FUNCTION_BLOCK FB_CommandTest EXTENDS TcUnit.FB_TestSuite
VAR
	sText			: STRING;
	iCounter		: INT;
END_VAR


T01_TestPoleceniaProstego ();
T02_TestPoleceniaZlozonego ();

METHOD PUBLIC MetodaDlaPolecenbiaProstego : bool
VAR_INPUT
END_VAR
THIS^.sText := 'jestem w tej metodzie';
iCounter := iCounter + 1;
MetodaDlaPolecenbiaProstego	:= FALSE;
END_METHOD

METHOD PROTECTED T01_TestPoleceniaProstego
VAR_INPUT
END_VAR
IF (TcUnit.TEST_ORDERED ('T01_TestPoleceniaProstego')) THEN
	GVL.fbCommandEasy.Test ();
	AssertTrue (Condition := GVL.fbCommandEasy.IsStatus (), 	Message := 'T01a - Bledny status');
	AssertFalse (Condition := GVL.fbCommandEasy.IsBusy (),		Message := 'T01b - Bledny stan');
	GVL.fbCommandEasy.Execute ();
	GVL.fbCommandEasy.Test ();
	AssertFalse (Condition := GVL.fbCommandEasy.IsStatus (), 	Message := 'T02a - Bledny status');
	AssertTrue (Condition := GVL.fbCommandEasy.IsBusy (),		Message := 'T02b - Bledny stan');
	
	GVL.fbCommandEasy.OperationExecute ();
	GVL.fbCommandEasy.Operation (bIN := MetodaDlaPolecenbiaProstego ());
	
	AssertTrue (Condition := GVL.fbCommandEasy.IsFirstCycle (),Message := 'T03a - Bledny stan pierwszego przejscia');
	AssertTrue (Condition := GVL.fbCommandEasy.IsLastCycle (),	Message := 'T03b - Bledny stan ostatniego przejscia');
	
	GVL.fbCommandEasy.OperationExecute ();
	
	AssertFalse (Condition := GVL.fbCommandEasy.IsFirstCycle (),	Message := 'T04a - Bledny stan pierwszego przejscia');
	AssertFalse (Condition := GVL.fbCommandEasy.IsLastCycle (),		Message := 'T04b - Bledny stan ostatniego przejscia');

	GVL.fbCommandEasy.OperationExecute ();
	
	AssertFalse (Condition := GVL.fbCommandEasy.IsLastCycle (),	Message := 'T05a - Bledny stan pierwszego przejscia');
	AssertTrue (Condition := GVL.fbCommandEasy.IsStatus (),		Message := 'T05b - Bledny stan statusy');
	
	TcUnit.TEST_FINISHED ();
END_IF
END_METHOD

METHOD PROTECTED T02_TestPoleceniaZlozonego : BOOL

VAR
	bResult: BOOL;
END_VAR
IF (TcUnit.TEST_ORDERED ('T02_TestPolecenia')) THEN
	GVL.fbCommand.Test ();
	AssertTrue (Condition := GVL.fbCommand.IsStatus (), 	Message := 'T01a - Bledny status');
	AssertFalse (Condition := GVL.fbCommand.IsBusy (),		Message := 'T01b - Bledny stan');
	
	GVL.fbCommand.Execute ();
	GVL.fbCommand.Test ();
	AssertFalse (Condition := GVL.fbCommand.IsStatus (), 	Message := 'T02a - Bledny status');
	AssertTrue (Condition := GVL.fbCommand.IsBusy (),		Message := 'T02b - Bledny stan');
	
	IF (GVL.fbCommand.OperationExecute ()) THEN;
		bResult				:= TRUE;
		GVL.fbCommand.Operation (bIN := GVL.fbCommand.CyklTestu ());
	ELSE
		bResult				:= FALSE;
	END_IF
	AssertTrue (Condition := GVL.fbCommand.IsFirstCycle (),Message := 'T03a - Bledny stan pierwszego przejscia');
	AssertFalse (Condition := GVL.fbCommand.IsLastCycle (),Message := 'T03b - Bledny stan ostatniego przejscia');
	AssertFalse (Condition := bResult, 						Message := 'T03c - Bledny wynik');
	
	IF (GVL.fbCommand.OperationExecute ()) THEN;
		bResult				:= TRUE;
		GVL.fbCommand.Operation (bIN := GVL.fbCommand.CyklTestu ());
	ELSE
		bResult				:= FALSE;
	END_IF
	AssertFalse (Condition := GVL.fbCommand.IsFirstCycle (),	Message := 'T04a - Bledny stan pierwszego przejscia');
	AssertFalse (Condition := GVL.fbCommand.IsLastCycle (),	Message := 'T04b - Bledny stan ostatniego przejscia');
	AssertTrue (Condition := bResult, 							Message := 'T04c - Bledny wynik');
	
	WRITE_PROTECTED_BOOL (Ptr := ADR (GVL.fbCommand.bFinish), Value := TRUE);
	IF (GVL.fbCommand.OperationExecute ()) THEN;
		bResult				:= TRUE;
		GVL.fbCommand.Operation (bIN := GVL.fbCommand.CyklTestu ());
	ELSE
		bResult				:= FALSE;
	END_IF
	AssertFalse (Condition := GVL.fbCommand.IsFirstCycle (),	Message := 'T05a - Bledny stan pierwszego przejscia');
	Asserttrue (Condition := GVL.fbCommand.IsLastCycle (),		Message := 'T05b - Bledny stan ostatniego przejscia');
	AssertTrue (Condition := bResult, 							Message := 'T05c - Bledny wynik');
	
	IF (GVL.fbCommand.OperationExecute ()) THEN;
		bResult				:= TRUE;
		GVL.fbCommand.Operation (bIN := GVL.fbCommand.CyklTestu ());
	ELSE
		bResult				:= FALSE;
	END_IF
	AssertFalse (Condition := GVL.fbCommand.IsFirstCycle (),	Message := 'T06a - Bledny stan pierwszego przejscia');
	AssertFalse (Condition := GVL.fbCommand.IsLastCycle (),	Message := 'T06b - Bledny stan ostatniego przejscia');
	AssertFalse (Condition := bResult, 							Message := 'T06c - Bledny wynik');

	

	TcUnit.TEST_FINISHED ();
END_IF
END_METHOD

END_FUNCTION_BLOCK

(* stored: Version 1.1.0.1, ProductVersion 3.1.4024.15
   POU FB_CommandTest: Id {20ace256-dafa-058e-3c0b-f94a17f6a90e}, SpecialFunc None
   Method MetodaDlaPolecenbiaProstego: Id {a3669c83-8900-0492-1d65-080f0e67aca3}
   Method T01_TestPoleceniaProstego: Id {189cc450-0321-4f98-954b-f6f385951fca}
   Method T02_TestPoleceniaZlozonego: Id {43608b7a-59c3-0e6c-3955-7f748c17b7f8} *)
